(* CODESYS project SignalSystem.project

Project tree, tasks and I/O mapping:
  Device : CODESYS Control Win V3 x64, 3S - Smart Software Solutions GmbH, version 3.5.9.50
    application Application
      libraries: Standard, * (System)
      task MainTask (cyclic, interval 4 ms, priority 0) calls EtherCAT_Master.EtherCAT_Task [EtherCAT_Master.EtherCAT_Task], PLC_PRG
      program PLC_PRG [LD]
      function block ThreeStateSignal [LD]
      Symbols
      function block OnOffDelay [ST]
      function block TrainDetection [ST]
    EtherCAT_Master : EtherCAT Master, 3S - Smart Software Solutions GmbH, version 3.5.9.50
        settings: MasterUseLRW = False; SlaveAutoRestart = False; NetworkName = 'ローカル エリア接続'; NetworkName = "ローカル エリア接続"; EnableTaskMessage = False; SyncOffset = 30; SrcAddress1 = 59546; SrcAddress2 = 2410977214
      NX_ECC202 : NX-ECC202 EtherCAT coupler V1.2, OMRON Corporation, order no. NX-ECC202, version Revision=16#00010002
          settings: Number of Outputs = 1; Number of Inputs = 5; Number of Infos about Outputs = 1; Number of Infos about Inputs = 5; StationAlias = 0; Sync.Length = 4; Sync.Length = 38; FMMU.Length = 4; FMMU.Length = 38; Number of RxPDOs of the Slave = 1; Number of TxPDOs of the Slave = 4; DC sync0 cycletime = 4000; DC sync1 cycletime = 4000; Number of SDO = 1; RxTxPdo.NumberofExcludes = 0; RxTxPdo.NumberofEntries = 1; RxTxPdo.Index = 16#1600; RxTxPdo.Fixed = True; RxTxPdo.Mandatory = True; RxTxPdo.Virtual = False; RxTxPdo.Sm = 2; RxTxPdo.Su = 0; RxTxPdo.Name = 'Output Data Set 1'; RxTxPdo.DependOnSlot = True; RxTxPdo.DependOnSlotGroup = False; NX_OD6121_5_1 Output Bit 32 bits.Index = 16#7003; NX_OD6121_5_1 Output Bit 32 bits.SubIndex = 1; NX_OD6121_5_1 Output Bit 32 bits.Size = 32; NX_OD6121_5_1 Output Bit 32 bits.Offset = 0; NX_OD6121_5_1 Output Bit 32 bits.DependOnSlot = True; NX_OD6121_5_1 Output Bit 32 bits.DependOnSlotGroup = True; RxTxPdo.NumberofExcludes = 0; RxTxPdo.NumberofEntries = 2; RxTxPdo.Index = 16#1BF8; RxTxPdo.Fixed = False; RxTxPdo.Mandatory = False; RxTxPdo.Virtual = False; RxTxPdo.Sm = 3; RxTxPdo.Su = 3; RxTxPdo.Name = '505th transmit PDO Mapping';
            RxTxPdo.DependOnSlot = False; RxTxPdo.DependOnSlotGroup = False; NX Unit Registration Status 125.Index = 16#3003; NX Unit Registration Status 125.SubIndex = 4; NX Unit Registration Status 125.Size = 128; NX Unit Registration Status 125.Offset = 0; NX Unit Registration Status 125.DependOnSlot = False; NX Unit Registration Status 125.DependOnSlotGroup = False; NX Unit I/O Data Active Status 125.Index = 16#3006; NX Unit I/O Data Active Status 125.SubIndex = 4; NX Unit I/O Data Active Status 125.Size = 128; NX Unit I/O Data Active Status 125.Offset = 0; NX Unit I/O Data Active Status 125.DependOnSlot = False; NX Unit I/O Data Active Status 125.DependOnSlotGroup = False; RxTxPdo.NumberofExcludes = 0; RxTxPdo.NumberofEntries = 1; RxTxPdo.Index = 16#1BFF; RxTxPdo.Fixed = True; RxTxPdo.Mandatory = False; RxTxPdo.Virtual = False; RxTxPdo.Sm = 3; RxTxPdo.Su = 3; RxTxPdo.Name = '512th transmit PDO Mapping'; RxTxPdo.DependOnSlot = False; RxTxPdo.DependOnSlotGroup = False; Sysmac Error Status.Index = 16#2002; Sysmac Error Status.SubIndex = 1; Sysmac Error Status.Size = 8; Sysmac Error Status.Offset = 0; Sysmac Error Status.DependOnSlot = False; Sysmac Error Status.DependOnSlotGroup = False; RxTxPdo.NumberofExcludes = 0; RxTxPdo.NumberofEntries = 1; RxTxPdo.Index = 16#1BF4; RxTxPdo.Fixed = True; RxTxPdo.Mandatory = False; RxTxPdo.Virtual = False; RxTxPdo.Sm = 3; RxTxPdo.Su = 3; RxTxPdo.Name = '501st transmit PDO Mapping';
            RxTxPdo.DependOnSlot = False; RxTxPdo.DependOnSlotGroup = False; Entry.Offset = 0; Entry.DependOnSlot = False; Entry.DependOnSlotGroup = False; RxTxPdo.NumberofExcludes = 0; RxTxPdo.NumberofEntries = 1; RxTxPdo.Index = 16#1A04; RxTxPdo.Fixed = True; RxTxPdo.Mandatory = True; RxTxPdo.Virtual = False; RxTxPdo.Sm = 3; RxTxPdo.Su = 0; RxTxPdo.Name = 'Input Data Set  1'; RxTxPdo.DependOnSlot = True; RxTxPdo.DependOnSlotGroup = False; NX_ID6142_5 Input Bit 32 bits.Index = 16#6023; NX_ID6142_5 Input Bit 32 bits.SubIndex = 1; NX_ID6142_5 Input Bit 32 bits.Size = 32; NX_ID6142_5 Input Bit 32 bits.Offset = 0; NX_ID6142_5 Input Bit 32 bits.DependOnSlot = True; NX_ID6142_5 Input Bit 32 bits.DependOnSlotGroup = True; NX_OD6121_5_1 Output Bit 32 bits.Name = 'NX_OD6121_5_1 Output Bit 32 bits'; NX_OD6121_5_1 Output Bit 32 bits.DataType = 'UDINT'; NX_OD6121_5_1 Output Bit 32 bits.Default = ''; NX_OD6121_5_1 Output Bit 32 bits.Comment = ''; NX Unit Registration Status 125.Name = 'NX Unit Registration Status 125'; NX Unit Registration Status 125.DataType = 'ARRAY [0..15] OF BYTE'; NX Unit Registration Status 125.Default = ''; NX Unit Registration Status 125.Comment = ''; NX Unit I/O Data Active Status 125.Name = 'NX Unit I/O Data Active Status 125'; NX Unit I/O Data Active Status 125.DataType = 'ARRAY [0..15] OF BYTE'; NX Unit I/O Data Active Status 125.Default = ''; NX Unit I/O Data Active Status 125.Comment = ''; Sysmac Error Status.Name = 'Sysmac Error Status'; Sysmac Error Status.DataType = 'USINT'; Sysmac Error Status.Default = ''; Sysmac Error Status.Comment = ''; Entry.Default = ''; NX_ID6142_5 Input Bit 32 bits.Name = 'NX_ID6142_5 Input Bit 32 bits';
            NX_ID6142_5 Input Bit 32 bits.DataType = 'UDINT'; NX_ID6142_5 Input Bit 32 bits.Default = ''; NX_ID6142_5 Input Bit 32 bits.Comment = ''
          unmapped channels: NX_OD6121_5_1 Output Bit 32 bits, NX Unit Registration Status 125, NX Unit I/O Data Active Status 125, Sysmac Error Status, , NX_ID6142_5 Input Bit 32 bits
        NX_ID6142_5 : General input, OMRON Corporation, order no. NX-ID6142-5, version 0
        NX_OD6121_5_1 : Tr.Out,32pts,NPN,12-24VDC,Free Run/IO Sync Refresh  ,ON 0.1ms,OFF 0.8ms, OMRON Corporation, order no. NX-OD6121-5, version 0
  data type E_SIGNAL_STATUS
*)

// E_SIGNAL_STATUS
TYPE E_SIGNAL_STATUS :
(
	R_Stop, YY_Warnig, Y_Caution, YG_Slowdown, G_Go
);
END_TYPE

// Device/Application/PLC_PRG
PROGRAM PLC_PRG
VAR
	IN0: BOOL;
	
	TrainDetectionExec: TrainDetection;
	abDetectSection: ARRAY[0..15] OF BOOL;
	
	Section0: ThreeStateSignal;
	Section1: ThreeStateSignal;
	Section2: ThreeStateSignal;
	Section3: ThreeStateSignal;
	
	eSignalStatus0: E_SIGNAL_STATUS;
	eSignalStatus1: E_SIGNAL_STATUS;
	eSignalStatus2: E_SIGNAL_STATUS;
	eSignalStatus3: E_SIGNAL_STATUS;
	
END_VAR

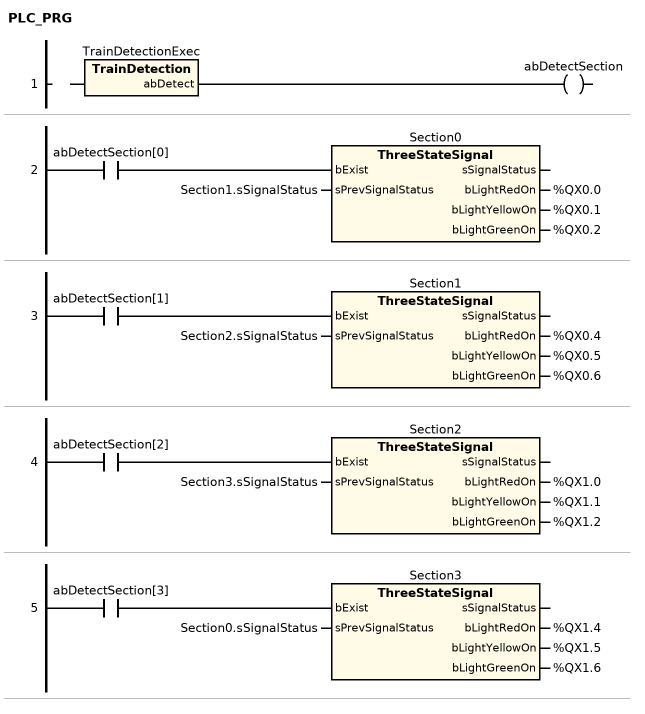
// NETWORK 1
TrainDetectionExec(); // TrainDetection
abDetectSection := TrainDetectionExec.abDetect;

// NETWORK 2
Section0(
    bExist := abDetectSection[0],
    sPrevSignalStatus := Section1.sSignalStatus,
    bLightRedOn => %QX0.0,
    bLightYellowOn => %QX0.1,
    bLightGreenOn => %QX0.2); // ThreeStateSignal

// NETWORK 3
Section1(
    bExist := abDetectSection[1],
    sPrevSignalStatus := Section2.sSignalStatus,
    bLightRedOn => %QX0.4,
    bLightYellowOn => %QX0.5,
    bLightGreenOn => %QX0.6); // ThreeStateSignal

// NETWORK 4
Section2(
    bExist := abDetectSection[2],
    sPrevSignalStatus := Section3.sSignalStatus,
    bLightRedOn => %QX1.0,
    bLightYellowOn => %QX1.1,
    bLightGreenOn => %QX1.2); // ThreeStateSignal

// NETWORK 5
Section3(
    bExist := abDetectSection[3],
    sPrevSignalStatus := Section0.sSignalStatus,
    bLightRedOn => %QX1.4,
    bLightYellowOn => %QX1.5,
    bLightGreenOn => %QX1.6); // ThreeStateSignal

END_PROGRAM

// Device/Application/TrainDetection
FUNCTION_BLOCK TrainDetection
VAR_INPUT
END_VAR
VAR_OUTPUT
	abDetect: ARRAY[0..15] OF BOOL;
END_VAR
VAR
	DetectDelayExec: ARRAY[0..15] OF OnOffDelay;
	dwIdx: INT;
END_VAR

DetectDelayExec[0](bIN := %IX36.0);
DetectDelayExec[1](bIN := %IX36.1);
DetectDelayExec[2](bIN := %IX36.2);
DetectDelayExec[3](bIN := %IX36.3);
DetectDelayExec[4](bIN := %IX36.4);
FOR dwIdx:=0 TO 15 DO
	abDetect[dwIdx] := DetectDelayExec[dwIdx].bOUT;
END_FOR

END_FUNCTION_BLOCK

// Device/Application/OnOffDelay
FUNCTION_BLOCK OnOffDelay
VAR_INPUT
	bIN: BOOL;
END_VAR
VAR_OUTPUT
	bOUT: BOOL;
END_VAR
VAR
	OffDelayTimer: Standard.TOF;
	OnDelayTimer: Standard.TON;
	bPrevOutput: BOOL;
END_VAR

OffDelayTimer(IN:=bIN, PT:=T#0.5S);
OnDelayTimer(IN:=bIN, PT:=T#0.5S);
IF bPrevOutput THEN
	bOUT := OffDelayTimer.Q;
ELSE
	bOUT := OnDelayTimer.Q;	
END_IF
bPrevOutput := bOUT;

END_FUNCTION_BLOCK

// Device/Application/ThreeStateSignal
FUNCTION_BLOCK ThreeStateSignal
VAR_INPUT
	bExist: BOOL;
	sPrevSignalStatus: E_SIGNAL_STATUS;
END_VAR
VAR_OUTPUT
	sSignalStatus: E_SIGNAL_STATUS;
	bLightRedOn: BOOL;
	bLightYellowOn: BOOL;
	bLightGreenOn: BOOL;
END_VAR
VAR
	// 内部補助接点
	bGreen0: BOOL;
	bGreen1: BOOL;
	bGreen2: BOOL;
	bGreen: BOOL;
END_VAR
VAR // added by the converter: edge detectors and wires of the graphical bodies
    _w1, _w2 : BOOL;
END_VAR

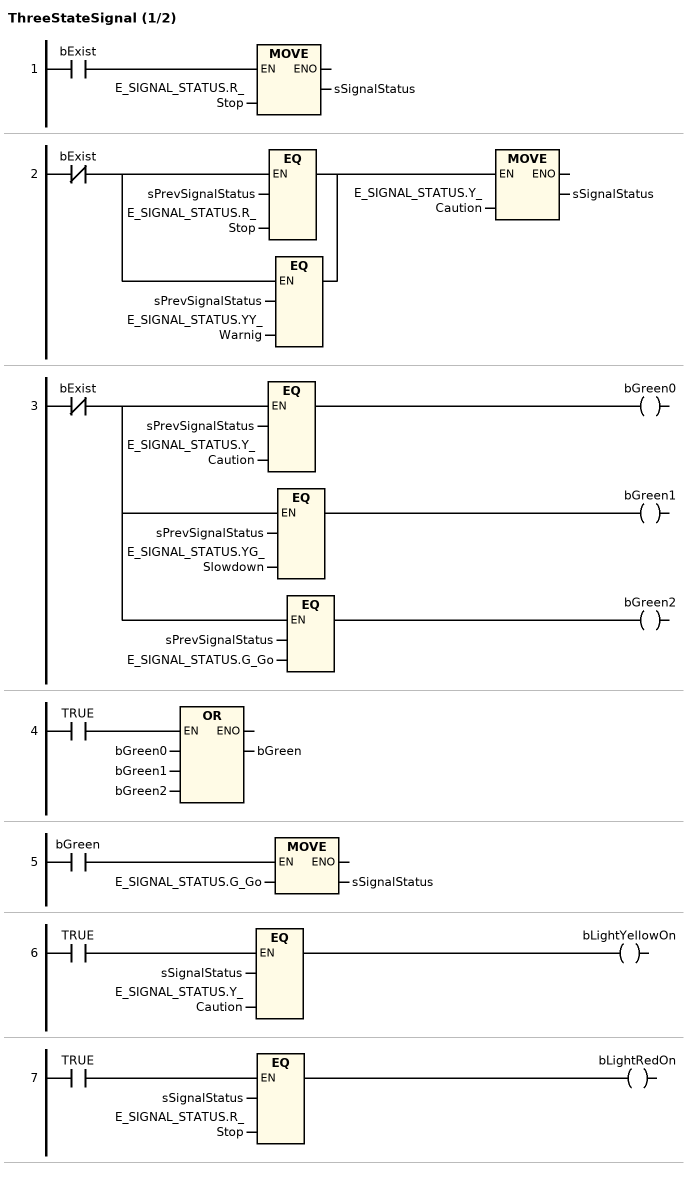
// NETWORK 1
IF bExist THEN sSignalStatus := E_SIGNAL_STATUS.R_Stop; END_IF

// NETWORK 2
_w1 := NOT bExist;
IF _w1 AND sPrevSignalStatus = E_SIGNAL_STATUS.R_Stop OR _w1 AND sPrevSignalStatus = E_SIGNAL_STATUS.YY_Warnig THEN
    sSignalStatus := E_SIGNAL_STATUS.Y_Caution;
END_IF

// NETWORK 3
_w2 := NOT bExist;
bGreen0 := _w2 AND sPrevSignalStatus = E_SIGNAL_STATUS.Y_Caution;
bGreen1 := _w2 AND sPrevSignalStatus = E_SIGNAL_STATUS.YG_Slowdown;
bGreen2 := _w2 AND sPrevSignalStatus = E_SIGNAL_STATUS.G_Go;

// NETWORK 4
bGreen := bGreen0 OR bGreen1 OR bGreen2;

// NETWORK 5
IF bGreen THEN sSignalStatus := E_SIGNAL_STATUS.G_Go; END_IF

// NETWORK 6
bLightYellowOn := sSignalStatus = E_SIGNAL_STATUS.Y_Caution;

// NETWORK 7
bLightRedOn := sSignalStatus = E_SIGNAL_STATUS.R_Stop;

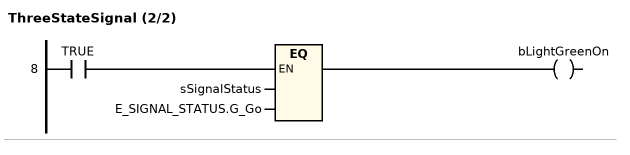
// NETWORK 8
bLightGreenOn := sSignalStatus = E_SIGNAL_STATUS.G_Go;

END_FUNCTION_BLOCK
